{attribute addProperty BoxType "EL3413-0000-0016"}
{attribute addProperty Id "STATUSAT %I*STATUS_3A9053451621CurrentAT %I*DINT32417VoltageAT %I*DINT32418Active_powerAT %I*DINT32419IndexAT %I*USINT8120Variant_valueAT %I*DINT32429"}
{attribute addProperty CRC "2680732136"}
{attribute addProperty SizeInBites "152"}
{attribute addProperty SizeInBytes "19"}
TYPE PM_Inputs_Channel_9FC8B9E8 :
STRUCT
	{attribute addProperty Name "STATUS"}
	STATUS AT %I* : STATUS_3A905345;
	{attribute addProperty Name "Current"}
	Current AT %I* : DINT;
	{attribute addProperty Name "Voltage"}
	Voltage AT %I* : DINT;
	{attribute addProperty Name "Active_power"}
	Active_power AT %I* : DINT;
	{attribute addProperty Name "Index"}
	Index AT %I* : USINT;
	{attribute addProperty Name "Variant_value"}
	Variant_value AT %I* : DINT;
END_STRUCT
END_TYPE

(* stored: Version 1.2.0.0, ProductVersion 3.1.4024.9
   DUT PM_Inputs_Channel_9FC8B9E8: Id {8a411a14-0525-4f29-a7dd-c3b197b2a433} *)
